{attribute 'qualified_only'}
{attribute 'strict'}
TYPE eXMCStateMachine :
(
	INIT,
	STOP,
	OP,
	ERROR
);
END_TYPE

(* stored: Version 1.1.0.1, ProductVersion 3.1.4024.12
   DUT eXMCStateMachine: Id {bc5173f6-f61a-4355-a022-66889dac662f} *)
